PROGRAM LD_Spantransportor
VAR
	Span_transportor: BOOL;
	Span_trans_Timer: TOF;
	Program_done: BOOL;
END_VAR

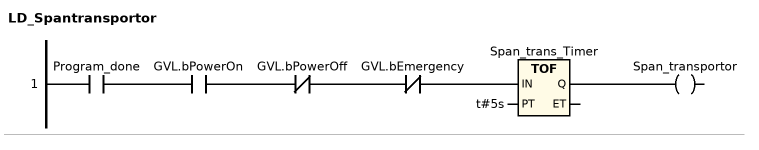
// NETWORK 1
Span_trans_Timer(IN := Program_done AND GVL.bPowerOn AND NOT GVL.bPowerOff AND NOT GVL.bEmergency, PT := t#5s); // TOF
Span_transportor := Span_trans_Timer.Q;

END_PROGRAM

(* stored: Version 1.1.0.1, ProductVersion 3.1.4024.10
   POU LD_Spantransportor: Id {6159a348-21ab-4f0d-9ec9-241d7cd48ad2}, SpecialFunc None *)
